{attribute 'qualified_only'}
{attribute 'strict'}
{attribute 'to_string'}
TYPE E_GripperControlOwner :
(
    None     := 0,
    Manual   := 10,
    Auto     := 20,
    Stop     := 30,
    Recovery := 40
);
END_TYPE

(* stored: Version 1.1.0.1, ProductVersion 3.1.4026.20
   DUT E_GripperControlOwner: Id {3fbe4961-775d-4a56-9e0c-96222375c2ba} *)
